FUNCTION_BLOCK TestAnyToString
VAR_INPUT
END_VAR
VAR_OUTPUT
END_VAR
VAR
  assert: FB_Assert('TestAnyToString');
END_VAR

assert.AbortAfterFail := TRUE;
CASE assert.State OF
16#0000:
  IF THIS^.transform_int_to_string() THEN
    assert.State := assert.State + 16#0010;
	END_IF
16#0010:
  IF THIS^.transform_real_to_string() THEN
    assert.State := assert.State + 16#0010;
	END_IF
16#0020:
  IF THIS^.transform_string_to_string() THEN
    assert.State := assert.State + 16#0010;
	END_IF
16#FFFF:
  ;
ELSE
  assert.PrintPassed('Done');
END_CASE

METHOD transform_int_to_string : BOOL
VAR_INPUT
END_VAR
VAR
  expected: STRING(10);
  actual: STRING(10);
  
  expected_int: INT;
END_VAR
expected_int := 300;
actual := _any_to_string(expected_int);
expected := '300';
transform_int_to_string := assert.AreEqualSTRING(expected, actual, 'Transform Int to String');
END_METHOD

METHOD transform_real_to_string : BOOL
VAR_INPUT
END_VAR
VAR
  expected: STRING(10);
  actual: STRING(10);
  
  expected_real: REAL;
END_VAR
expected_real := 123.456;
actual := _any_to_string(expected_real);
expected := '123.456';
transform_real_to_string := assert.AreEqualSTRING(expected, actual, 'Transform Real to String');
END_METHOD

METHOD transform_string_to_string : BOOL
VAR_INPUT
END_VAR
VAR
  expected: STRING(10);
  actual: STRING(10);
END_VAR
expected := 'foobar';
actual := _any_to_string(expected);
transform_string_to_string := assert.AreEqualSTRING(expected, actual, 'Transform String to String');
END_METHOD

END_FUNCTION_BLOCK

(* stored: Version 1.1.0.1, ProductVersion 3.1.4022.7
   POU TestAnyToString: Id {e3f564dd-9d1b-4c17-bf9f-2a4db2a30ec0}, SpecialFunc None
   Method transform_int_to_string: Id {0b0c21a9-66ff-4830-9de5-e116677f2c88}
   Method transform_real_to_string: Id {490a3233-c267-4c89-87f8-0049a24e8d1a}
   Method transform_string_to_string: Id {4523adc2-8204-4fe8-a9c7-eb6c28aefc54} *)
